PROGRAM MAIN
VAR
	nstep:INT:=20;
	connection:FB_sqlcommandevt(snetid:='', tTimeout:=T#5S);
	
	Datareturn:fb_datareturn;
	createtable:fb_createtable;
	insertRecord:fb_insertrecord;
	WriteCSV: fb_CSVWrite;
	ReadCSV:fb_CSVRead;
	
	st_insertdata:ST_insertdata;
	bDataReturn:BOOL:=FALSE;
	bCreateTable:BOOL:=FALSE;
	bInsert:BOOL:=FALSE;
	
	dbid:UINT:=3;
	table:STRING:='$'1_kamra$'';
	start:STRING:='$'2020-07-01 15:00:01$'';
	end:STRING:='$'2020-08-30 15:00:01$'';
	
END_VAR

CASE nstep OF 
	
	20:
		IF bdatareturn THEN
			datareturn.ClearArray();
			nstep:=30;
			bdatareturn:=FALSE;
		END_IF
		IF bCreateTable THEN
			nstep:=40;
			bcreatetable:=FALSE;
		END_IF
		IF bInsert THEN
			nstep:=50;
			bInsert:=FALSE;
		END_IF
		
		
		
	30:	// datareturn
		
		datareturn(dbid:=dbid,
					table:=table,
					start:=start,
					end:=end,
					bexecute:=TRUE);
		IF datareturn.Error THEN
			nstep:=99;
		ELSE
		IF datareturn.bReady THEN
			
			nstep:=20;
			datareturn.Reset();
		END_IF
		END_IF
		
	40:	//create table
		createtable(table:=table,
					bExecute:=TRUE,
					DBID:=dbid);
		IF createtable.bError THEN
			nstep:=99;
		ELSE	
		IF createtable.bReady THEN
			createtable.Reset();	
			nstep:=20;
		END_IF
		END_IF
	50: // insert data
		//st_insertData.Datum:='$'2020-01-01 12:00:20$'';//DT#2020-07-28-15:00:01 ;
		////st_insertdata.hum_act:='1';
		//st_insertdata.hum_set:='2';
		//st_insertdata.temp_act:='3';
		//st_insertdata.temp_set:='4';
		insertrecord(insertdata:=st_insertdata,
					table:=table,
					DBID:=dbid,
					bExecute:=TRUE);
		IF insertrecord.bError THEN
			nstep:=99;
		ELSE
		IF insertrecord.bReady THEN
			nstep:=20;
			insertrecord.Reset();
		END_IF
		END_IF

	60: // write csv
		st_insertData.Datum:='2020-01-01 12:00:20';//DT#2020-07-28-15:00:01 ;
		st_insertdata.hum_act:='1';
		st_insertdata.hum_set:='2';
		st_insertdata.temp_act:='3';
		st_insertdata.temp_set:='4';
		WriteCSV(dbid:=4,
				table:='1_kamra',
				bExecute:=TRUE);
		IF WriteCSV.bError THEN
			nstep:=99;
		ELSE
		IF  WriteCSV.bReady THEN
			nstep:=20;
			WriteCSV.reset();
		END_IF
		END_IF		
	
	70:	//ReadCSV
		ReadCSV(dbid:=4,
				table:='1_kamra',
				bExecute:=TRUE);
		IF ReadCSV.bError THEN
			nstep:=99;
		ELSE
		IF  ReadCSV.bReady THEN
			nstep:=20;
			ReadCSV.reset();
		END_IF
		END_IF		
	99:// error
		;	
			
END_CASE

END_PROGRAM

(* stored: Version 1.1.0.1, ProductVersion 3.1.4024.2
   POU MAIN: Id {4d934eb9-7ebd-4818-b7fc-5be66a99ea54}, SpecialFunc None *)
